// TIA Portal V18 export
FUNCTION "DIvars" : Void   // FC10008, LAD
{ S7_Optimized_Access := 'TRUE' }
VERSION : 0.1
// stored: AutoNumber false, IsIECCheckEnabled false, SetENOAutomatically false, UDAEnableTagReadback false
   VAR_INPUT
      xInput : Bool;
      iFuncSystem : Byte;
      iFuncVar : Byte;
   END_VAR
BEGIN

REGION Network 1 (SCL)
   CASE #iFuncSystem OF
       0:  // Statement section case 2 to 4
           ;
       1..4:  // Statement section case 1
           CASE #iFuncVar OF
               0:  // 
                   ;
               1:  // 
                   "AHUDI".DI.xHeaterPumpReady[#iFuncSystem] := #xInput;
               2:  // 
                   "AHUDI".DI.xHeaterPumpInd[#iFuncSystem] := #xInput;
               3:  // 
                   "AHUDI".DI.xHeaterPumpAlarm[#iFuncSystem] := #xInput;
               4:  // 
                   "AHUDI".DI.xSAFAnalogReady[#iFuncSystem] := #xInput;
               5:  // 
                   "AHUDI".DI.xSAFAnalogInd[#iFuncSystem] := #xInput;
               6:  // 
                   "AHUDI".DI.xSAFAnalogAlarm[#iFuncSystem] := #xInput;
               7:  // 
                   "AHUDI".DI.xSAFSp1Ready[#iFuncSystem] := #xInput;
               8:  // 
                   "AHUDI".DI.xSAFSp1Ind[#iFuncSystem] := #xInput;
               9:  // 
                   "AHUDI".DI.xSAFSp1Alarm[#iFuncSystem] := #xInput;
               10:  // 
                   "AHUDI".DI.xSAFSp2Ready[#iFuncSystem] := #xInput;
               11:  // 
                   "AHUDI".DI.xSAFSp2Ind[#iFuncSystem] := #xInput;
               12:  // 
                   "AHUDI".DI.xSAFSp2Alarm[#iFuncSystem] := #xInput;
               13:  // 
                   "AHUDI".DI.xSAFdPInd[#iFuncSystem] := #xInput;
               14:  // 
                   "AHUDI".DI.xFrostProtTstat[#iFuncSystem] := #xInput;
               15:  // 
                   "AHUDI".DI.xSAFdPAlarm[#iFuncSystem] := #xInput;
               16:  // 
                   "AHUDI".DI.xSAFPanelSelectorOff[#iFuncSystem] := #xInput;
               17:  // 
                   "AHUDI".DI.xSAFPanelSelector1St[#iFuncSystem] := #xInput;
               18:  // 
                   "AHUDI".DI.xSAFPanelSelector2St[#iFuncSystem] := #xInput;
               19:  // 
                   "AHUDI".DI.xSAFPanelSelectorAuto[#iFuncSystem] := #xInput;
               20:  //
                   "AHUDI".DI.xSAFMotorPTCAlarm[#iFuncSystem] := #xInput;
               21:  //
                   "AHUDI".DI.xServiceSwitchOnAHU[#iFuncSystem] := #xInput;
               22:  //
                   "AHUDI".DI.xCoolerAlarm[#iFuncSystem] := #xInput;
               23:  //
                   "AHUDI".DI.xCoolerC1Ind[#iFuncSystem] := #xInput;
               24:  //
                   "AHUDI".DI.xCoolerC2Ind[#iFuncSystem] := #xInput;
               25:  //
                   "AHUDI".DI.xFilterdP[#iFuncSystem] := #xInput;
               26:  //
                   "AHUDI".DI.xHeaterPumpModeInAuto[#iFuncSystem] := #xInput;
               ELSE
                   ;
           END_CASE;
       5..9:
           ;
       10:  //    
           CASE #iFuncVar OF
               0:  //
                   ;
               1:
                   "HCsDI".Requests.xHCPump1Ready[1] := #xInput;
               2:
                   "HCsDI".Requests.xHCPump1Ind[1] := #xInput;
               3: //    
                   "HCsDI".Requests.xHCPump1Alarm[1] := #xInput;
               4:  //
                   "HCsDI".Requests.xHCPump2Ready[1] := #xInput;
               5:  //
                   "HCsDI".Requests.xHCPump2Ind[1] := #xInput;
               6:  //
                   "HCsDI".Requests.xHCPump2Alarm[1] := #xInput;
               7:  //
                   "HCsDI".Requests.xHCDoublePumpInAuto[1] := #xInput;
               8:
                   "HCsDI".Requests.xHCPump1Ready[2] := #xInput;
               9:
                   "HCsDI".Requests.xHCPump1Ind[2] := #xInput;
               10: //    
                   "HCsDI".Requests.xHCPump1Alarm[2] := #xInput;
               11:  //
                   "HCsDI".Requests.xHCPump2Ready[2] := #xInput;
               12:  //
                   "HCsDI".Requests.xHCPump2Ind[2] := #xInput;
               13:  //
                   "HCsDI".Requests.xHCPump2Alarm[2] := #xInput;
               14:  //
                   "HCsDI".Requests.xHCDoublePumpInAuto[2] := #xInput;
               15..20: //
                   ;
               21:  //
                   "HSsDI".Requests.xBoilerShuntPumpReady[1] := #xInput;
               22:  //
                   "HSsDI".Requests.xBoilerShuntPumpInd[1] := #xInput;
               23:  //
                   "HSsDI".Requests.xBoilerShuntPumpAlarm[1] := #xInput;
               24:  //
                   "HSsDI".Requests.xBoilerShuntPumpInAuto[1] := #xInput;
               25:  //
                   "HSsDI".Requests.xBoilerStage1Ind[1] := #xInput;
               26:  //
                   "HSsDI".Requests.xBoilerStage2Ind[1] := #xInput;
               27:  //
                   "HSsDI".Requests.xBurnerAlarm[1] := #xInput;
               28:  //
                   "HSsDI".Requests.xBoilerAlarm[1] := #xInput;
               29:  //
                   "HSsDI".Requests.xBoilerReady[1] := #xInput;
               30:  //
                   "HSsDI".Requests.xBoilerReserve[1] := #xInput;
               31:  //
                   "HSsDI".Requests.xBoilerShuntPumpReady[2] := #xInput;
               32:  //
                   "HSsDI".Requests.xBoilerShuntPumpInd[2] := #xInput;
               33:  //
                   "HSsDI".Requests.xBoilerShuntPumpAlarm[2] := #xInput;
               34:  //
                   "HSsDI".Requests.xBoilerShuntPumpInAuto[2] := #xInput;
               35:  //
                   "HSsDI".Requests.xBoilerStage1Ind[2] := #xInput;
               36:  //
                   "HSsDI".Requests.xBoilerStage2Ind[2] := #xInput;
               37:  //
                   "HSsDI".Requests.xBurnerAlarm[2] := #xInput;
               38:  //
                   "HSsDI".Requests.xBoilerAlarm[2] := #xInput;
               39:  //
                   "HSsDI".Requests.xBoilerReady[2] := #xInput;
               40:  //
                   "HSsDI".Requests.xBoilerReserve[2] := #xInput;
               41:
                   "HSsDI".Requests.xSeasonWinter[1] := #xInput;
               42:
                   "HSsDI".Requests.xSeasonSummer[1] := #xInput;
               43:
                   "HSsDI".Requests.xSeasonAuto[1] := #xInput;
               44:
                   "HSsDI".Requests.xSeasonWinter[2] := #xInput;
               45:
                   "HSsDI".Requests.xSeasonSummer[2] := #xInput;
               46:
                   "HSsDI".Requests.xSeasonAuto[2] := #xInput;
               47..50:
                   ;
               51:
                   "HSsDI".Requests.xBoilerWaterLvl[1] := #xInput;
               52:
                   "HSsDI".Requests.xBoilerPmin[1] := #xInput;
               53:
                   "HSsDI".Requests.xBoilerPmax[1] := #xInput;
               54..60:
                   ;
               61:
                   "HSsDI".Requests.xBoilerWaterLvl[2] := #xInput;
               62:
                   "HSsDI".Requests.xBoilerPmin[2] := #xInput;
               63:
                   "HSsDI".Requests.xBoilerPmax[2] := #xInput;
               ELSE
                   ;
           END_CASE;
       11..20:
           ;
       21:
           CASE #iFuncVar OF
           0:
               ;
           1..8:
               "AHUProxyCH".Vars.xCHRlyIsOnInd[#iFuncVar] := #xInput;
           9..16:
               "AHUProxyCH".Vars.xCHRlyIsOffInd[#iFuncVar] := #xInput;
           ELSE
               ;
           END_CASE;
       22..99:
           ;
       100:
           CASE #iFuncVar OF
               0:
                   ;
               1:
                   "DLsDI".Requests.xDieselLineHeatingReady[1] := #xInput;
               2:
                   "DLsDI".Requests.xDieselLineHeatingReady[2] := #xInput;
               3:
                   "DLsDI".Requests.xDieselLineHeatingInd[1]:= #xInput;
               4:
                   "DLsDI".Requests.xDieselLineHeatingInd[2] := #xInput;
               5:
                   "DLsDI".Requests.xDieselLinePumpInd[1] := #xInput;
               6:
                   "DLsDI".Requests.xDieselLinePumpInd[2]:= #xInput;
               7:
                   "DLsDI".Requests.xDieselLinePnom := #xInput;
               8:
                   "DLsDI".Requests.xDieselLineValveToBoilerInd := #xInput;
               9:
                   "DLsDI".Requests.xDieselLinePmax:= #xInput;
               10:
                   "DLsDI".Requests.xDieselLinePumpZoneWaterFloodAlarm := #xInput;
               11:
                   "DLsDI".Requests.xDieselLineMainTankDoubleWallAlarmInd := #xInput;
               12:
                   "DLsDI".Requests.xDieselLineMainTankMinLevelInd:= #xInput;
               13:
                   "DLsDI".Requests.Reserve1 := #xInput;
               14:
                   "DLsDI".Requests.Reserve2 := #xInput;
               15:
                   "DLsDI".Requests.xDieselLinePumpPanelSelectorOff:= #xInput;
               16:
                   "DLsDI".Requests.xDieselLinePumpPanelSelectorP1Man := #xInput;
               17:
                   "DLsDI".Requests.xDieselLinePumpPanelSelectorP2Man := #xInput;
               18:
                   "DLsDI".Requests.xDieselLinePumpPanelSelectorAuto:= #xInput;
               ELSE
                   ;
           END_CASE;
       ELSE  // Statement section ELSE
           ;
   END_CASE;
END_REGION
END_FUNCTION
